FUNCTION_BLOCK FB_TMO_LED
VAR_INPUT
	iTermBits : UINT;
	
	{attribute 'pytmc' := '
        pv: CIL:PCT
        field: EGU %
    '}
	fIlluminatorPercent : LREAL;
END_VAR
VAR
	iIlluminatorINT AT %Q*: INT;

    {attribute 'pytmc' := '
        pv: PWR
        field: ZNAM OFF
        field: ONAM ON
    '}
    bLedPower AT %Q*: BOOL;

//    fIlluminatorPercent: LREAL;
//    fbGetIllPercent: FB_AnalogInput;
    fbSetIllPercent: FB_AnalogOutput;

    bLedInit: BOOL := FALSE;
END_VAR

// Turn the LED off by default
(*
IF not bLedInit THEN
    bLedPower := FALSE;
//    bLedInit := TRUE;
END_IF
*)

// Illuminator conversion to percentage
fbSetIllPercent(
    fReal:=fIlluminatorPercent,
    fSafeMax:=100,
    fSafeMin:=0,
    iTermBits:=iTermBits,
    fTermMax:=100,
    fTermMin:=0,
    iRaw=>iIlluminatorINT);

IF  fIlluminatorPercent > 0 THEN
	bLedPower := TRUE;
ELSE
	bLEDPower := FALSE;
END_IF

(*	
fbGetIllPercent(
    iRaw:=iIlluminatorINT,
    iTermBits:=15,
    fTermMax:=100,
    fTermMin:=0,
    fReal=>fIlluminatorPercent);
*)

END_FUNCTION_BLOCK

(* stored: Version 1.1.0.1, ProductVersion 3.1.4022.18
   POU FB_TMO_LED: Id {a99d7fba-0318-482f-b028-cab96116f8cb}, SpecialFunc None *)
